// TIA Portal V21 export
TYPE "StrutturaComando"
   STRUCT
      Selezione : Int;   // 0 = Forced Off 1 = Manual 2= Auto
      Stato : Int;   // 1 = Off 2 = On 3 = Fault 4 = Forced On 5 = Forced Off
      Man : Bool;
      Auto : Bool;
      OFF : Bool;
      ON : Bool;
   END_STRUCT;
END_TYPE
